PROGRAM PRG_TXI_VAC_VALVES
VAR
END_VAR

fb_PC1K3_VGC_01(
    i_stUSG := fb_PC1K3_PIP_02.q_IG,
    i_stDSG := fb_PC1K3_PIP_01.q_IG,
    i_xDis_DPIlk := FALSE,
    i_xEPS_OK := TRUE,
    i_xPMPS_OK := TRUE,
    i_xExt_OK := TRUE,
    i_xOverrideMode := xSystemOverrideMode1, 
    io_fbFFHWO := g_FastFaultOutput1, 
    fbArbiter := fbArbiter1
); 

fb_TV1K3_VGC_01(
    i_stUSG := fb_PC1K3_PIP_02.q_IG,
    i_stDSG := fb_PC1K3_PIP_01.q_IG,
    i_xDis_DPIlk := FALSE,
    i_xEPS_OK := TRUE,
    i_xPMPS_OK := TRUE,
    i_xExt_OK := TRUE,
    i_xOverrideMode := xSystemOverrideMode1, 
    io_fbFFHWO := g_FastFaultOutput1, 
    fbArbiter := fbArbiter1
);

END_PROGRAM

(* stored: Version 1.1.0.1, ProductVersion 3.1.4024.6
   POU PRG_TXI_VAC_VALVES: Id {4c9a7319-3f14-4d3b-bb2f-4b6392242f38}, SpecialFunc None *)
